PROGRAM MAIN
VAR
	fb_ReadInputs : ModbusReadInputs;
	fb_WriteOutputs : ModbusWriteOutputs;
	data: ARRAY [0..1] OF BYTE;
	bSensorEndConveyor: BOOL;
	bStartStopConveyor: ARRAY [0..1] OF BYTE := [2#0000_0001, 2#0000_0000];
END_VAR

fb_ReadInputs(Data=> data);
bSensorEndConveyor := data[0].0;

IF bSensorEndConveyor THEN
	fb_WriteOutputs(Data := CONTROL.StartConveyor);
//ELSIF NOT bSensorEndConveyor THEN
	//fb_WriteOutputs(Data := CONTROL.StopConveyor);	
END_IF;

END_PROGRAM

(* stored: Version 1.1.0.1, ProductVersion 3.1.4024.9
   POU MAIN: Id {46a88e70-018e-4a2c-8074-d59c6124b5c0}, SpecialFunc None *)
